RoboDK station: CNC_LATHE.rdk

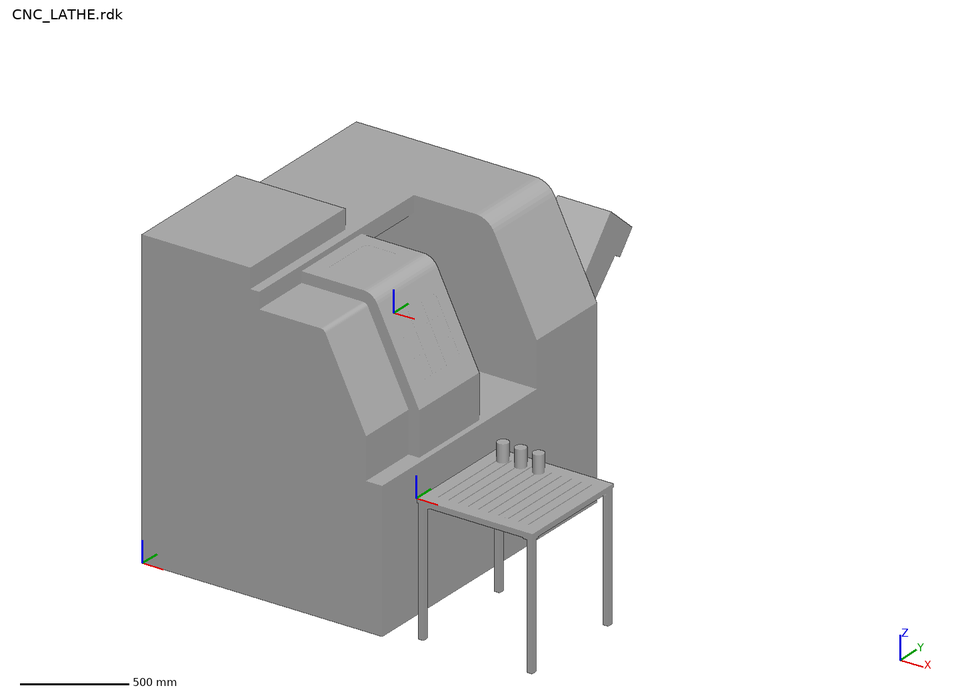
[picture v0: the station drawn from its stored meshes, robots at their saved joint values, targets as dots, program paths as lines]
Station CNC_LATHE (saved by RoboDK 5.1.1). Poses are relative to the parent item; angles as X-Y-Z fixed-axis rotations.
  - frame Marco_Estacion at (0, 0, 0) mm
    - object CNC at (-1290, 1630, 1260) mm, size 2146.6 x 2360 x 1680 mm, geometry from Ensamblaje1.stl
    - frame Marco_Mesa at (1490, 70, 720) mm
      - object Cilinder1 at (100, 550, 0) mm, size 60 x 60 x 100 mm, geometry from Cilinder.stl
      - object Cilinder2 at (200, 550, 0) mm, size 60 x 60 x 100 mm, geometry from Cilinder.stl
      - object Cilinder3 at (300, 550, 0) mm, size 60 x 60 x 100 mm, geometry from Cilinder.stl
    - frame Marco_Mandril at (850, 800, 1200) mm
  - program Reacomodar_Objetos (1 instructions, listed below)

--- program Reacomodar_Objetos ---
  Reemplazar objetos
